ABB RobotStudio station: Obelix2_20190227-112918.rsstn

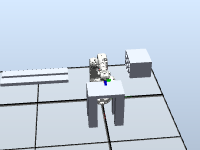
Station Obelix2 (saved by RobotStudio 6.8.8148.134)
Controller IRB_140T_6kg_0.81m
  mechanical unit ROB_1: IRB140T_6_81_C_03, 6 joints, base frame (0, 0, 0) mm
Layout (positions relative to the parent item):
  - IRB140T_6_81_C_03 [mechanism, from Robots\IRB140T_6_81_C_G_03.rslib] at (0, 0, 0) mm; joint values [0, 0, 0, 0, 0.5236, 0] (rad or m)
  - conveyor [part]
  - ManipulationTable [part]
  - conveyor_2 [part]
  - Oven_2 [part]
Targets, tools, work objects and paths stored in the station, written as RAPID:
! task T_ROB1
MODULE Module1
  CONST robtarget pHome:=[[506.291650772,0,679.49999918],[0.499999994,0,0.866025407,0],[0,0,0,0],[9E+09,9E+09,9E+09,9E+09,9E+09,9E+09]];
ENDMODULE

